// TIA Portal V18 export
// export: Created 2024-02-15T13:16:19.4089202Z, ExportSetting WithDefaults, DisplayName Totally Integrated Automation Portal, DisplayVersion V18 Update 3, DisplayName TIA Portal Openness, DisplayVersion V18 Update 3, DisplayName TIA Portal Version Control Interface, DisplayVersion V18, DisplayName TIA Portal Test Suite Advanced, DisplayVersion V18, DisplayName SINAMICS Startdrive Advanced, DisplayVersion V18, DisplayName SINAMICS Startdrive G130, G150, S120, S150, SINAMICS MV, S210, DisplayVersion V18, DisplayName SINAMICS Startdrive G110M, G120, G120C, G120D, G120P, G115D, DisplayVersion V18, DisplayName STEP 7 Professional, DisplayVersion V18 Update 3, DisplayName STEP 7 CFC, DisplayVersion V18, DisplayName STEP 7 Safety, DisplayVersion V18, DisplayName WinCC Advanced / Unified PC, DisplayVersion V18 Update 3, DisplayName SIMATIC Visualization Architect, DisplayVersion V18 Update 3
FUNCTION "COM_8864079" : Void   // FC36, LAD
{ S7_Optimized_Access := 'TRUE' }
VERSION : 0.1
// stored: AutoNumber true, IsIECCheckEnabled false, SetENOAutomatically false, UDAEnableTagReadback false
   VAR_TEMP   // added for the SCL form of the ladder/FBD networks
      _w1 : Bool;
   END_VAR
BEGIN

REGION Network 1: Echange avec API SDM Demande de Froid
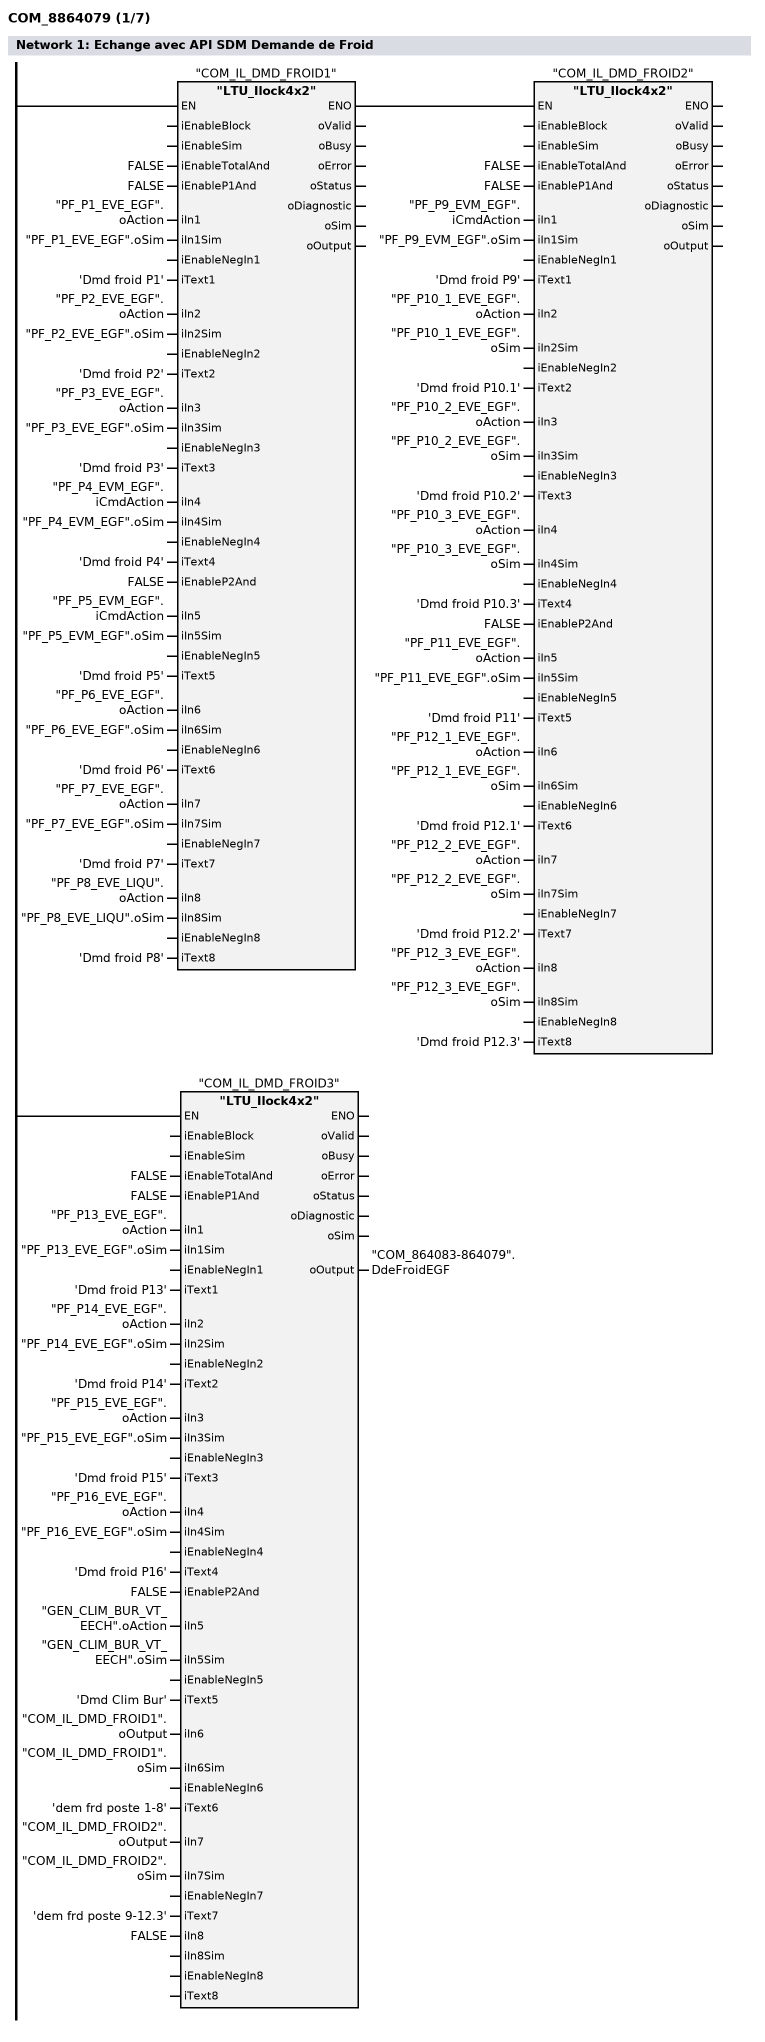
   RUNG wire#powerrail
      "COM_IL_DMD_FROID1"(iEnableBlock :=, iEnableSim :=, iEnableTotalAnd := FALSE, iEnableP1And := FALSE, iIn1 := "PF_P1_EVE_EGF".oAction, iIn1Sim := "PF_P1_EVE_EGF".oSim, iEnableNegIn1 :=, iText1 := 'Dmd froid P1', iIn2 := "PF_P2_EVE_EGF".oAction, iIn2Sim := "PF_P2_EVE_EGF".oSim, iEnableNegIn2 :=, iText2 := 'Dmd froid P2', iIn3 := "PF_P3_EVE_EGF".oAction, iIn3Sim := "PF_P3_EVE_EGF".oSim, iEnableNegIn3 :=, iText3 := 'Dmd froid P3', iIn4 := "PF_P4_EVM_EGF".iCmdAction, iIn4Sim := "PF_P4_EVM_EGF".oSim, iEnableNegIn4 :=, iText4 := 'Dmd froid P4', iEnableP2And := FALSE, iIn5 := "PF_P5_EVM_EGF".iCmdAction, iIn5Sim := "PF_P5_EVM_EGF".oSim, iEnableNegIn5 :=, iText5 := 'Dmd froid P5', iIn6 := "PF_P6_EVE_EGF".oAction, iIn6Sim := "PF_P6_EVE_EGF".oSim, iEnableNegIn6 :=, iText6 := 'Dmd froid P6', iIn7 := "PF_P7_EVE_EGF".oAction, iIn7Sim := "PF_P7_EVE_EGF".oSim, iEnableNegIn7 :=, iText7 := 'Dmd froid P7', iIn8 := "PF_P8_EVE_LIQU".oAction, iIn8Sim := "PF_P8_EVE_LIQU".oSim, iEnableNegIn8 :=, iText8 := 'Dmd froid P8', oValid =>, oBusy =>, oError =>, oStatus =>, oDiagnostic =>, oSim =>, oOutput =>)
      "COM_IL_DMD_FROID2"(iEnableBlock :=, iEnableSim :=, iEnableTotalAnd := FALSE, iEnableP1And := FALSE, iIn1 := "PF_P9_EVM_EGF".iCmdAction, iIn1Sim := "PF_P9_EVM_EGF".oSim, iEnableNegIn1 :=, iText1 := 'Dmd froid P9', iIn2 := "PF_P10_1_EVE_EGF".oAction, iIn2Sim := "PF_P10_1_EVE_EGF".oSim, iEnableNegIn2 :=, iText2 := 'Dmd froid P10.1', iIn3 := "PF_P10_2_EVE_EGF".oAction, iIn3Sim := "PF_P10_2_EVE_EGF".oSim, iEnableNegIn3 :=, iText3 := 'Dmd froid P10.2', iIn4 := "PF_P10_3_EVE_EGF".oAction, iIn4Sim := "PF_P10_3_EVE_EGF".oSim, iEnableNegIn4 :=, iText4 := 'Dmd froid P10.3', iEnableP2And := FALSE, iIn5 := "PF_P11_EVE_EGF".oAction, iIn5Sim := "PF_P11_EVE_EGF".oSim, iEnableNegIn5 :=, iText5 := 'Dmd froid P11', iIn6 := "PF_P12_1_EVE_EGF".oAction, iIn6Sim := "PF_P12_1_EVE_EGF".oSim, iEnableNegIn6 :=, iText6 := 'Dmd froid P12.1', iIn7 := "PF_P12_2_EVE_EGF".oAction, iIn7Sim := "PF_P12_2_EVE_EGF".oSim, iEnableNegIn7 :=, iText7 := 'Dmd froid P12.2', iIn8 := "PF_P12_3_EVE_EGF".oAction, iIn8Sim := "PF_P12_3_EVE_EGF".oSim, iEnableNegIn8 :=, iText8 := 'Dmd froid P12.3', oValid =>, oBusy =>, oError =>, oStatus =>, oDiagnostic =>, oSim =>, oOutput =>)
   END_RUNG
   RUNG wire#powerrail
      "COM_IL_DMD_FROID3"(iEnableBlock :=, iEnableSim :=, iEnableTotalAnd := FALSE, iEnableP1And := FALSE, iIn1 := "PF_P13_EVE_EGF".oAction, iIn1Sim := "PF_P13_EVE_EGF".oSim, iEnableNegIn1 :=, iText1 := 'Dmd froid P13', iIn2 := "PF_P14_EVE_EGF".oAction, iIn2Sim := "PF_P14_EVE_EGF".oSim, iEnableNegIn2 :=, iText2 := 'Dmd froid P14', iIn3 := "PF_P15_EVE_EGF".oAction, iIn3Sim := "PF_P15_EVE_EGF".oSim, iEnableNegIn3 :=, iText3 := 'Dmd froid P15', iIn4 := "PF_P16_EVE_EGF".oAction, iIn4Sim := "PF_P16_EVE_EGF".oSim, iEnableNegIn4 :=, iText4 := 'Dmd froid P16', iEnableP2And := FALSE, iIn5 := "GEN_CLIM_BUR_VT_EECH".oAction, iIn5Sim := "GEN_CLIM_BUR_VT_EECH".oSim, iEnableNegIn5 :=, iText5 := 'Dmd Clim Bur', iIn6 := "COM_IL_DMD_FROID1".oOutput, iIn6Sim := "COM_IL_DMD_FROID1".oSim, iEnableNegIn6 :=, iText6 := 'dem frd poste 1-8', iIn7 := "COM_IL_DMD_FROID2".oOutput, iIn7Sim := "COM_IL_DMD_FROID2".oSim, iEnableNegIn7 :=, iText7 := 'dem frd poste 9-12.3', iIn8 := FALSE, iIn8Sim :=, iEnableNegIn8 :=, iText8 :=, oValid =>, oBusy =>, oError =>, oStatus =>, oDiagnostic =>, oSim =>, oOutput => "COM_864083-864079".DdeFroidEGF)
   END_RUNG
   // the same network as SCL:
   "COM_IL_DMD_FROID1"(iEnableTotalAnd := FALSE,   // "LTU_Ilock4x2"
                       iEnableP1And := FALSE,
                       iIn1 := "PF_P1_EVE_EGF".oAction,
                       iIn1Sim := "PF_P1_EVE_EGF".oSim,
                       iText1 := 'Dmd froid P1',
                       iIn2 := "PF_P2_EVE_EGF".oAction,
                       iIn2Sim := "PF_P2_EVE_EGF".oSim,
                       iText2 := 'Dmd froid P2',
                       iIn3 := "PF_P3_EVE_EGF".oAction,
                       iIn3Sim := "PF_P3_EVE_EGF".oSim,
                       iText3 := 'Dmd froid P3',
                       iIn4 := "PF_P4_EVM_EGF".iCmdAction,
                       iIn4Sim := "PF_P4_EVM_EGF".oSim,
                       iText4 := 'Dmd froid P4',
                       iEnableP2And := FALSE,
                       iIn5 := "PF_P5_EVM_EGF".iCmdAction,
                       iIn5Sim := "PF_P5_EVM_EGF".oSim,
                       iText5 := 'Dmd froid P5',
                       iIn6 := "PF_P6_EVE_EGF".oAction,
                       iIn6Sim := "PF_P6_EVE_EGF".oSim,
                       iText6 := 'Dmd froid P6',
                       iIn7 := "PF_P7_EVE_EGF".oAction,
                       iIn7Sim := "PF_P7_EVE_EGF".oSim,
                       iText7 := 'Dmd froid P7',
                       iIn8 := "PF_P8_EVE_LIQU".oAction,
                       iIn8Sim := "PF_P8_EVE_LIQU".oSim,
                       iText8 := 'Dmd froid P8',
                       ENO => #_w1);
   IF #_w1 THEN
       "COM_IL_DMD_FROID2"(iEnableTotalAnd := FALSE,   // "LTU_Ilock4x2"
                           iEnableP1And := FALSE,
                           iIn1 := "PF_P9_EVM_EGF".iCmdAction,
                           iIn1Sim := "PF_P9_EVM_EGF".oSim,
                           iText1 := 'Dmd froid P9',
                           iIn2 := "PF_P10_1_EVE_EGF".oAction,
                           iIn2Sim := "PF_P10_1_EVE_EGF".oSim,
                           iText2 := 'Dmd froid P10.1',
                           iIn3 := "PF_P10_2_EVE_EGF".oAction,
                           iIn3Sim := "PF_P10_2_EVE_EGF".oSim,
                           iText3 := 'Dmd froid P10.2',
                           iIn4 := "PF_P10_3_EVE_EGF".oAction,
                           iIn4Sim := "PF_P10_3_EVE_EGF".oSim,
                           iText4 := 'Dmd froid P10.3',
                           iEnableP2And := FALSE,
                           iIn5 := "PF_P11_EVE_EGF".oAction,
                           iIn5Sim := "PF_P11_EVE_EGF".oSim,
                           iText5 := 'Dmd froid P11',
                           iIn6 := "PF_P12_1_EVE_EGF".oAction,
                           iIn6Sim := "PF_P12_1_EVE_EGF".oSim,
                           iText6 := 'Dmd froid P12.1',
                           iIn7 := "PF_P12_2_EVE_EGF".oAction,
                           iIn7Sim := "PF_P12_2_EVE_EGF".oSim,
                           iText7 := 'Dmd froid P12.2',
                           iIn8 := "PF_P12_3_EVE_EGF".oAction,
                           iIn8Sim := "PF_P12_3_EVE_EGF".oSim,
                           iText8 := 'Dmd froid P12.3');
   END_IF;
   "COM_IL_DMD_FROID3"(iEnableTotalAnd := FALSE,   // "LTU_Ilock4x2"
                       iEnableP1And := FALSE,
                       iIn1 := "PF_P13_EVE_EGF".oAction,
                       iIn1Sim := "PF_P13_EVE_EGF".oSim,
                       iText1 := 'Dmd froid P13',
                       iIn2 := "PF_P14_EVE_EGF".oAction,
                       iIn2Sim := "PF_P14_EVE_EGF".oSim,
                       iText2 := 'Dmd froid P14',
                       iIn3 := "PF_P15_EVE_EGF".oAction,
                       iIn3Sim := "PF_P15_EVE_EGF".oSim,
                       iText3 := 'Dmd froid P15',
                       iIn4 := "PF_P16_EVE_EGF".oAction,
                       iIn4Sim := "PF_P16_EVE_EGF".oSim,
                       iText4 := 'Dmd froid P16',
                       iEnableP2And := FALSE,
                       iIn5 := "GEN_CLIM_BUR_VT_EECH".oAction,
                       iIn5Sim := "GEN_CLIM_BUR_VT_EECH".oSim,
                       iText5 := 'Dmd Clim Bur',
                       iIn6 := "COM_IL_DMD_FROID1".oOutput,
                       iIn6Sim := "COM_IL_DMD_FROID1".oSim,
                       iText6 := 'dem frd poste 1-8',
                       iIn7 := "COM_IL_DMD_FROID2".oOutput,
                       iIn7Sim := "COM_IL_DMD_FROID2".oSim,
                       iText7 := 'dem frd poste 9-12.3',
                       iIn8 := FALSE,
                       oOutput => "COM_864083-864079".DdeFroidEGF);
END_REGION

REGION Network 2: Echange avec API SDM Demande de Dégivrage
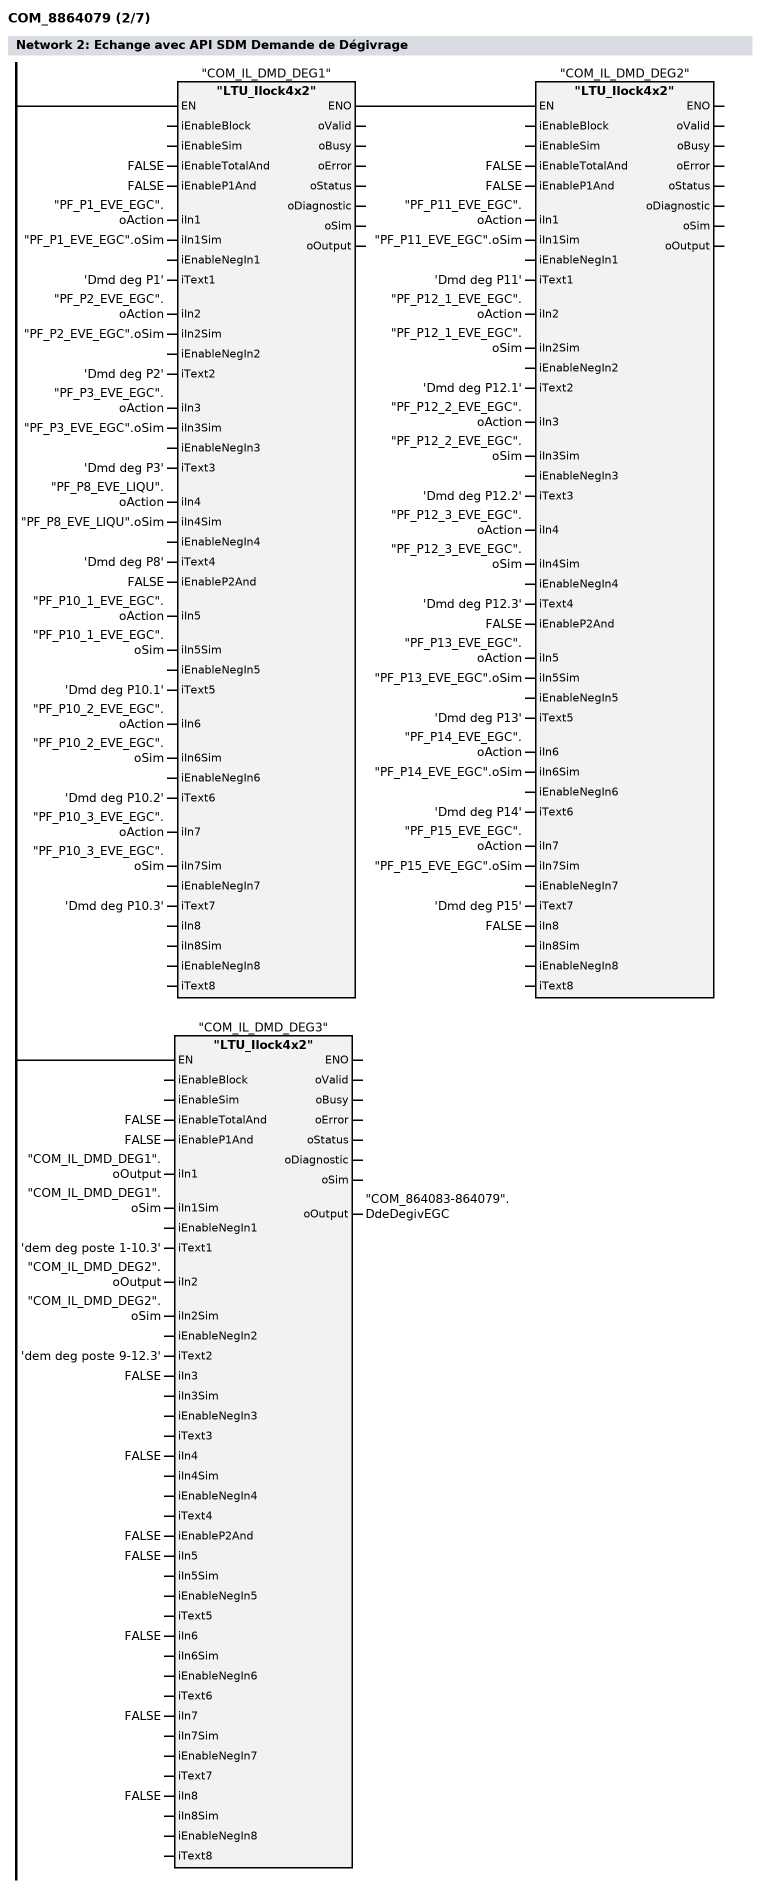
   RUNG wire#powerrail
      "COM_IL_DMD_DEG1"(iEnableBlock :=, iEnableSim :=, iEnableTotalAnd := FALSE, iEnableP1And := FALSE, iIn1 := "PF_P1_EVE_EGC".oAction, iIn1Sim := "PF_P1_EVE_EGC".oSim, iEnableNegIn1 :=, iText1 := 'Dmd deg P1', iIn2 := "PF_P2_EVE_EGC".oAction, iIn2Sim := "PF_P2_EVE_EGC".oSim, iEnableNegIn2 :=, iText2 := 'Dmd deg P2', iIn3 := "PF_P3_EVE_EGC".oAction, iIn3Sim := "PF_P3_EVE_EGC".oSim, iEnableNegIn3 :=, iText3 := 'Dmd deg P3', iIn4 := "PF_P8_EVE_LIQU".oAction, iIn4Sim := "PF_P8_EVE_LIQU".oSim, iEnableNegIn4 :=, iText4 := 'Dmd deg P8', iEnableP2And := FALSE, iIn5 := "PF_P10_1_EVE_EGC".oAction, iIn5Sim := "PF_P10_1_EVE_EGC".oSim, iEnableNegIn5 :=, iText5 := 'Dmd deg P10.1', iIn6 := "PF_P10_2_EVE_EGC".oAction, iIn6Sim := "PF_P10_2_EVE_EGC".oSim, iEnableNegIn6 :=, iText6 := 'Dmd deg P10.2', iIn7 := "PF_P10_3_EVE_EGC".oAction, iIn7Sim := "PF_P10_3_EVE_EGC".oSim, iEnableNegIn7 :=, iText7 := 'Dmd deg P10.3', iIn8 :=, iIn8Sim :=, iEnableNegIn8 :=, iText8 :=, oValid =>, oBusy =>, oError =>, oStatus =>, oDiagnostic =>, oSim =>, oOutput =>)
      "COM_IL_DMD_DEG2"(iEnableBlock :=, iEnableSim :=, iEnableTotalAnd := FALSE, iEnableP1And := FALSE, iIn1 := "PF_P11_EVE_EGC".oAction, iIn1Sim := "PF_P11_EVE_EGC".oSim, iEnableNegIn1 :=, iText1 := 'Dmd deg P11', iIn2 := "PF_P12_1_EVE_EGC".oAction, iIn2Sim := "PF_P12_1_EVE_EGC".oSim, iEnableNegIn2 :=, iText2 := 'Dmd deg P12.1', iIn3 := "PF_P12_2_EVE_EGC".oAction, iIn3Sim := "PF_P12_2_EVE_EGC".oSim, iEnableNegIn3 :=, iText3 := 'Dmd deg P12.2', iIn4 := "PF_P12_3_EVE_EGC".oAction, iIn4Sim := "PF_P12_3_EVE_EGC".oSim, iEnableNegIn4 :=, iText4 := 'Dmd deg P12.3', iEnableP2And := FALSE, iIn5 := "PF_P13_EVE_EGC".oAction, iIn5Sim := "PF_P13_EVE_EGC".oSim, iEnableNegIn5 :=, iText5 := 'Dmd deg P13', iIn6 := "PF_P14_EVE_EGC".oAction, iIn6Sim := "PF_P14_EVE_EGC".oSim, iEnableNegIn6 :=, iText6 := 'Dmd deg P14', iIn7 := "PF_P15_EVE_EGC".oAction, iIn7Sim := "PF_P15_EVE_EGC".oSim, iEnableNegIn7 :=, iText7 := 'Dmd deg P15', iIn8 := FALSE, iIn8Sim :=, iEnableNegIn8 :=, iText8 :=, oValid =>, oBusy =>, oError =>, oStatus =>, oDiagnostic =>, oSim =>, oOutput =>)
   END_RUNG
   RUNG wire#powerrail
      "COM_IL_DMD_DEG3"(iEnableBlock :=, iEnableSim :=, iEnableTotalAnd := FALSE, iEnableP1And := FALSE, iIn1 := "COM_IL_DMD_DEG1".oOutput, iIn1Sim := "COM_IL_DMD_DEG1".oSim, iEnableNegIn1 :=, iText1 := 'dem deg poste 1-10.3', iIn2 := "COM_IL_DMD_DEG2".oOutput, iIn2Sim := "COM_IL_DMD_DEG2".oSim, iEnableNegIn2 :=, iText2 := 'dem deg poste 9-12.3', iIn3 := FALSE, iIn3Sim :=, iEnableNegIn3 :=, iText3 :=, iIn4 := FALSE, iIn4Sim :=, iEnableNegIn4 :=, iText4 :=, iEnableP2And := FALSE, iIn5 := FALSE, iIn5Sim :=, iEnableNegIn5 :=, iText5 :=, iIn6 := FALSE, iIn6Sim :=, iEnableNegIn6 :=, iText6 :=, iIn7 := FALSE, iIn7Sim :=, iEnableNegIn7 :=, iText7 :=, iIn8 := FALSE, iIn8Sim :=, iEnableNegIn8 :=, iText8 :=, oValid =>, oBusy =>, oError =>, oStatus =>, oDiagnostic =>, oSim =>, oOutput => "COM_864083-864079".DdeDegivEGC)
   END_RUNG
   // the same network as SCL:
   "COM_IL_DMD_DEG1"(iEnableTotalAnd := FALSE,   // "LTU_Ilock4x2"
                     iEnableP1And := FALSE,
                     iIn1 := "PF_P1_EVE_EGC".oAction,
                     iIn1Sim := "PF_P1_EVE_EGC".oSim,
                     iText1 := 'Dmd deg P1',
                     iIn2 := "PF_P2_EVE_EGC".oAction,
                     iIn2Sim := "PF_P2_EVE_EGC".oSim,
                     iText2 := 'Dmd deg P2',
                     iIn3 := "PF_P3_EVE_EGC".oAction,
                     iIn3Sim := "PF_P3_EVE_EGC".oSim,
                     iText3 := 'Dmd deg P3',
                     iIn4 := "PF_P8_EVE_LIQU".oAction,
                     iIn4Sim := "PF_P8_EVE_LIQU".oSim,
                     iText4 := 'Dmd deg P8',
                     iEnableP2And := FALSE,
                     iIn5 := "PF_P10_1_EVE_EGC".oAction,
                     iIn5Sim := "PF_P10_1_EVE_EGC".oSim,
                     iText5 := 'Dmd deg P10.1',
                     iIn6 := "PF_P10_2_EVE_EGC".oAction,
                     iIn6Sim := "PF_P10_2_EVE_EGC".oSim,
                     iText6 := 'Dmd deg P10.2',
                     iIn7 := "PF_P10_3_EVE_EGC".oAction,
                     iIn7Sim := "PF_P10_3_EVE_EGC".oSim,
                     iText7 := 'Dmd deg P10.3',
                     ENO => #_w1);
   IF #_w1 THEN
       "COM_IL_DMD_DEG2"(iEnableTotalAnd := FALSE,   // "LTU_Ilock4x2"
                         iEnableP1And := FALSE,
                         iIn1 := "PF_P11_EVE_EGC".oAction,
                         iIn1Sim := "PF_P11_EVE_EGC".oSim,
                         iText1 := 'Dmd deg P11',
                         iIn2 := "PF_P12_1_EVE_EGC".oAction,
                         iIn2Sim := "PF_P12_1_EVE_EGC".oSim,
                         iText2 := 'Dmd deg P12.1',
                         iIn3 := "PF_P12_2_EVE_EGC".oAction,
                         iIn3Sim := "PF_P12_2_EVE_EGC".oSim,
                         iText3 := 'Dmd deg P12.2',
                         iIn4 := "PF_P12_3_EVE_EGC".oAction,
                         iIn4Sim := "PF_P12_3_EVE_EGC".oSim,
                         iText4 := 'Dmd deg P12.3',
                         iEnableP2And := FALSE,
                         iIn5 := "PF_P13_EVE_EGC".oAction,
                         iIn5Sim := "PF_P13_EVE_EGC".oSim,
                         iText5 := 'Dmd deg P13',
                         iIn6 := "PF_P14_EVE_EGC".oAction,
                         iIn6Sim := "PF_P14_EVE_EGC".oSim,
                         iText6 := 'Dmd deg P14',
                         iIn7 := "PF_P15_EVE_EGC".oAction,
                         iIn7Sim := "PF_P15_EVE_EGC".oSim,
                         iText7 := 'Dmd deg P15',
                         iIn8 := FALSE);
   END_IF;
   "COM_IL_DMD_DEG3"(iEnableTotalAnd := FALSE,   // "LTU_Ilock4x2"
                     iEnableP1And := FALSE,
                     iIn1 := "COM_IL_DMD_DEG1".oOutput,
                     iIn1Sim := "COM_IL_DMD_DEG1".oSim,
                     iText1 := 'dem deg poste 1-10.3',
                     iIn2 := "COM_IL_DMD_DEG2".oOutput,
                     iIn2Sim := "COM_IL_DMD_DEG2".oSim,
                     iText2 := 'dem deg poste 9-12.3',
                     iIn3 := FALSE,
                     iIn4 := FALSE,
                     iEnableP2And := FALSE,
                     iIn5 := FALSE,
                     iIn6 := FALSE,
                     iIn7 := FALSE,
                     iIn8 := FALSE,
                     oOutput => "COM_864083-864079".DdeDegivEGC);
END_REGION

REGION Network 3: Echange avec API SDM Défaut prioritaire AGBT1
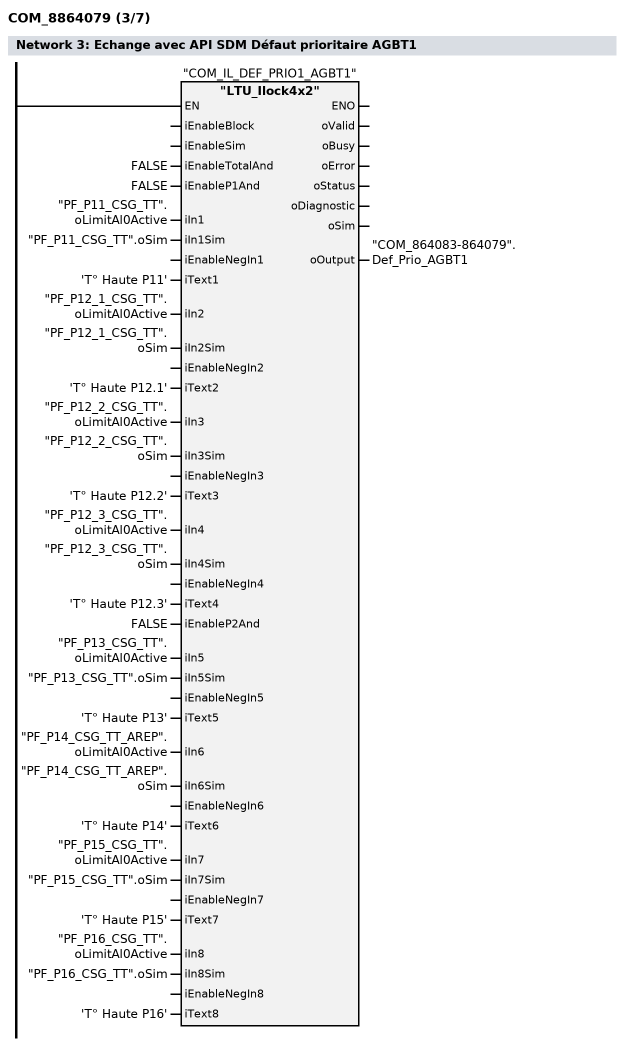
   RUNG wire#powerrail
      "COM_IL_DEF_PRIO1_AGBT1"(iEnableBlock :=, iEnableSim :=, iEnableTotalAnd := FALSE, iEnableP1And := FALSE, iIn1 := "PF_P11_CSG_TT".oLimitAl0Active, iIn1Sim := "PF_P11_CSG_TT".oSim, iEnableNegIn1 :=, iText1 := 'T° Haute P11', iIn2 := "PF_P12_1_CSG_TT".oLimitAl0Active, iIn2Sim := "PF_P12_1_CSG_TT".oSim, iEnableNegIn2 :=, iText2 := 'T° Haute P12.1', iIn3 := "PF_P12_2_CSG_TT".oLimitAl0Active, iIn3Sim := "PF_P12_2_CSG_TT".oSim, iEnableNegIn3 :=, iText3 := 'T° Haute P12.2', iIn4 := "PF_P12_3_CSG_TT".oLimitAl0Active, iIn4Sim := "PF_P12_3_CSG_TT".oSim, iEnableNegIn4 :=, iText4 := 'T° Haute P12.3', iEnableP2And := FALSE, iIn5 := "PF_P13_CSG_TT".oLimitAl0Active, iIn5Sim := "PF_P13_CSG_TT".oSim, iEnableNegIn5 :=, iText5 := 'T° Haute P13', iIn6 := "PF_P14_CSG_TT_AREP".oLimitAl0Active, iIn6Sim := "PF_P14_CSG_TT_AREP".oSim, iEnableNegIn6 :=, iText6 := 'T° Haute P14', iIn7 := "PF_P15_CSG_TT".oLimitAl0Active, iIn7Sim := "PF_P15_CSG_TT".oSim, iEnableNegIn7 :=, iText7 := 'T° Haute P15', iIn8 := "PF_P16_CSG_TT".oLimitAl0Active, iIn8Sim := "PF_P16_CSG_TT".oSim, iEnableNegIn8 :=, iText8 := 'T° Haute P16', oValid =>, oBusy =>, oError =>, oStatus =>, oDiagnostic =>, oSim =>, oOutput => "COM_864083-864079".Def_Prio_AGBT1)
   END_RUNG
   // the same network as SCL:
   "COM_IL_DEF_PRIO1_AGBT1"(iEnableTotalAnd := FALSE,   // "LTU_Ilock4x2"
                           iEnableP1And := FALSE,
                           iIn1 := "PF_P11_CSG_TT".oLimitAl0Active,
                           iIn1Sim := "PF_P11_CSG_TT".oSim,
                           iText1 := 'T° Haute P11',
                           iIn2 := "PF_P12_1_CSG_TT".oLimitAl0Active,
                           iIn2Sim := "PF_P12_1_CSG_TT".oSim,
                           iText2 := 'T° Haute P12.1',
                           iIn3 := "PF_P12_2_CSG_TT".oLimitAl0Active,
                           iIn3Sim := "PF_P12_2_CSG_TT".oSim,
                           iText3 := 'T° Haute P12.2',
                           iIn4 := "PF_P12_3_CSG_TT".oLimitAl0Active,
                           iIn4Sim := "PF_P12_3_CSG_TT".oSim,
                           iText4 := 'T° Haute P12.3',
                           iEnableP2And := FALSE,
                           iIn5 := "PF_P13_CSG_TT".oLimitAl0Active,
                           iIn5Sim := "PF_P13_CSG_TT".oSim,
                           iText5 := 'T° Haute P13',
                           iIn6 := "PF_P14_CSG_TT_AREP".oLimitAl0Active,
                           iIn6Sim := "PF_P14_CSG_TT_AREP".oSim,
                           iText6 := 'T° Haute P14',
                           iIn7 := "PF_P15_CSG_TT".oLimitAl0Active,
                           iIn7Sim := "PF_P15_CSG_TT".oSim,
                           iText7 := 'T° Haute P15',
                           iIn8 := "PF_P16_CSG_TT".oLimitAl0Active,
                           iIn8Sim := "PF_P16_CSG_TT".oSim,
                           iText8 := 'T° Haute P16',
                           oOutput => "COM_864083-864079".Def_Prio_AGBT1);
END_REGION

REGION Network 4: Echange avec API SDM Défaut NON prioritaire AGBT1
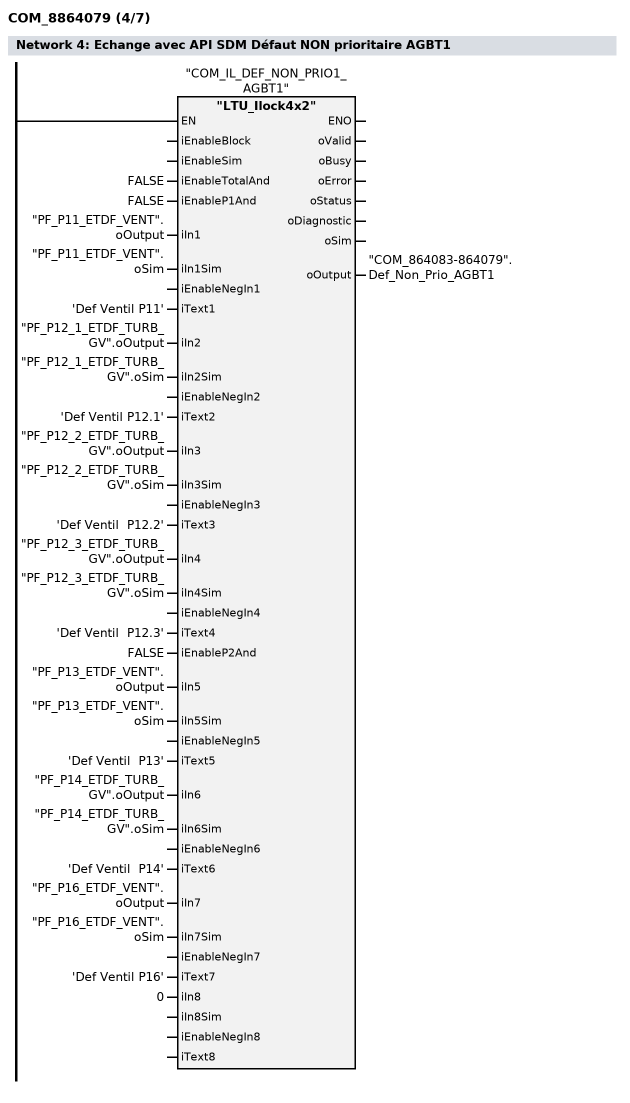
   RUNG wire#powerrail
      "COM_IL_DEF_NON_PRIO1_AGBT1"(iEnableBlock :=, iEnableSim :=, iEnableTotalAnd := FALSE, iEnableP1And := FALSE, iIn1 := "PF_P11_ETDF_VENT".oOutput, iIn1Sim := "PF_P11_ETDF_VENT".oSim, iEnableNegIn1 :=, iText1 := 'Def Ventil P11', iIn2 := "PF_P12_1_ETDF_TURB_GV".oOutput, iIn2Sim := "PF_P12_1_ETDF_TURB_GV".oSim, iEnableNegIn2 :=, iText2 := 'Def Ventil P12.1', iIn3 := "PF_P12_2_ETDF_TURB_GV".oOutput, iIn3Sim := "PF_P12_2_ETDF_TURB_GV".oSim, iEnableNegIn3 :=, iText3 := 'Def Ventil  P12.2', iIn4 := "PF_P12_3_ETDF_TURB_GV".oOutput, iIn4Sim := "PF_P12_3_ETDF_TURB_GV".oSim, iEnableNegIn4 :=, iText4 := 'Def Ventil  P12.3', iEnableP2And := FALSE, iIn5 := "PF_P13_ETDF_VENT".oOutput, iIn5Sim := "PF_P13_ETDF_VENT".oSim, iEnableNegIn5 :=, iText5 := 'Def Ventil  P13', iIn6 := "PF_P14_ETDF_TURB_GV".oOutput, iIn6Sim := "PF_P14_ETDF_TURB_GV".oSim, iEnableNegIn6 :=, iText6 := 'Def Ventil  P14', iIn7 := "PF_P16_ETDF_VENT".oOutput, iIn7Sim := "PF_P16_ETDF_VENT".oSim, iEnableNegIn7 :=, iText7 := 'Def Ventil P16', iIn8 := 0, iIn8Sim :=, iEnableNegIn8 :=, iText8 :=, oValid =>, oBusy =>, oError =>, oStatus =>, oDiagnostic =>, oSim =>, oOutput => "COM_864083-864079".Def_Non_Prio_AGBT1)
   END_RUNG
   // the same network as SCL:
   "COM_IL_DEF_NON_PRIO1_AGBT1"(iEnableTotalAnd := FALSE,   // "LTU_Ilock4x2"
                           iEnableP1And := FALSE,
                           iIn1 := "PF_P11_ETDF_VENT".oOutput,
                           iIn1Sim := "PF_P11_ETDF_VENT".oSim,
                           iText1 := 'Def Ventil P11',
                           iIn2 := "PF_P12_1_ETDF_TURB_GV".oOutput,
                           iIn2Sim := "PF_P12_1_ETDF_TURB_GV".oSim,
                           iText2 := 'Def Ventil P12.1',
                           iIn3 := "PF_P12_2_ETDF_TURB_GV".oOutput,
                           iIn3Sim := "PF_P12_2_ETDF_TURB_GV".oSim,
                           iText3 := 'Def Ventil  P12.2',
                           iIn4 := "PF_P12_3_ETDF_TURB_GV".oOutput,
                           iIn4Sim := "PF_P12_3_ETDF_TURB_GV".oSim,
                           iText4 := 'Def Ventil  P12.3',
                           iEnableP2And := FALSE,
                           iIn5 := "PF_P13_ETDF_VENT".oOutput,
                           iIn5Sim := "PF_P13_ETDF_VENT".oSim,
                           iText5 := 'Def Ventil  P13',
                           iIn6 := "PF_P14_ETDF_TURB_GV".oOutput,
                           iIn6Sim := "PF_P14_ETDF_TURB_GV".oSim,
                           iText6 := 'Def Ventil  P14',
                           iIn7 := "PF_P16_ETDF_VENT".oOutput,
                           iIn7Sim := "PF_P16_ETDF_VENT".oSim,
                           iText7 := 'Def Ventil P16',
                           iIn8 := 0,
                           oOutput => "COM_864083-864079".Def_Non_Prio_AGBT1);
END_REGION

REGION Network 5: Echange avec API SDM Défaut prioritaire AGBT2
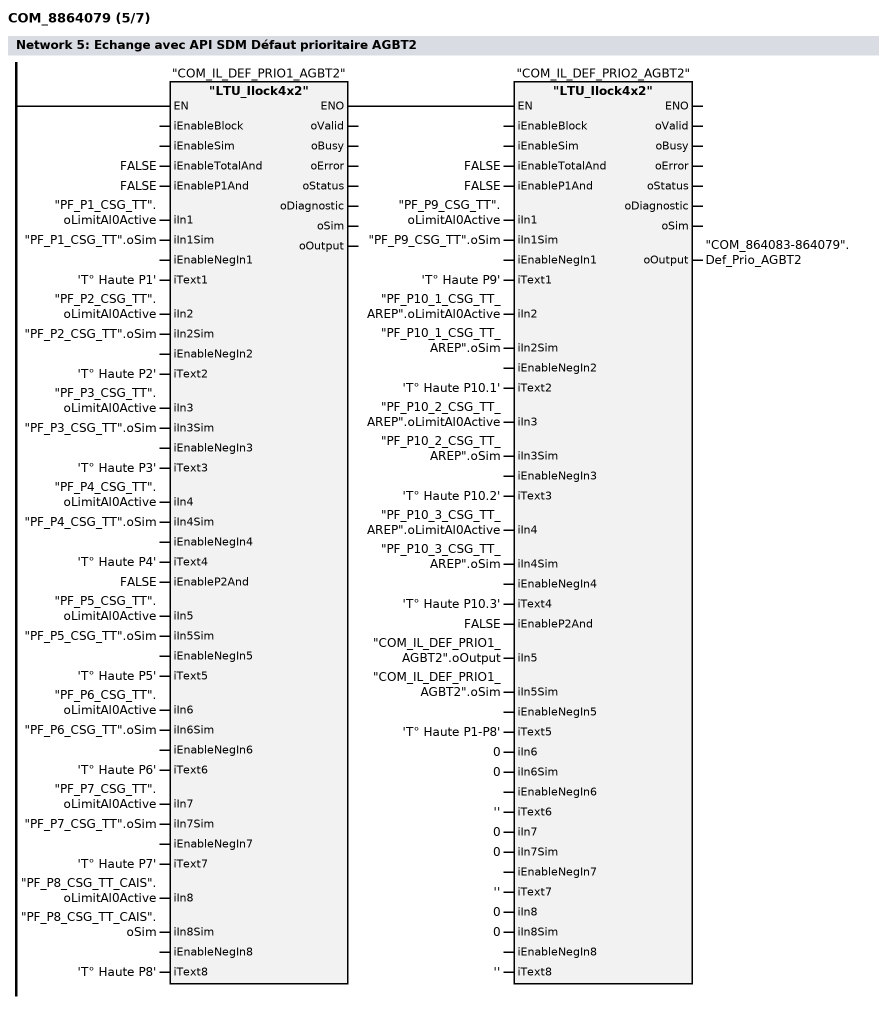
   RUNG wire#powerrail
      "COM_IL_DEF_PRIO1_AGBT2"(iEnableBlock :=, iEnableSim :=, iEnableTotalAnd := FALSE, iEnableP1And := FALSE, iIn1 := "PF_P1_CSG_TT".oLimitAl0Active, iIn1Sim := "PF_P1_CSG_TT".oSim, iEnableNegIn1 :=, iText1 := 'T° Haute P1', iIn2 := "PF_P2_CSG_TT".oLimitAl0Active, iIn2Sim := "PF_P2_CSG_TT".oSim, iEnableNegIn2 :=, iText2 := 'T° Haute P2', iIn3 := "PF_P3_CSG_TT".oLimitAl0Active, iIn3Sim := "PF_P3_CSG_TT".oSim, iEnableNegIn3 :=, iText3 := 'T° Haute P3', iIn4 := "PF_P4_CSG_TT".oLimitAl0Active, iIn4Sim := "PF_P4_CSG_TT".oSim, iEnableNegIn4 :=, iText4 := 'T° Haute P4', iEnableP2And := FALSE, iIn5 := "PF_P5_CSG_TT".oLimitAl0Active, iIn5Sim := "PF_P5_CSG_TT".oSim, iEnableNegIn5 :=, iText5 := 'T° Haute P5', iIn6 := "PF_P6_CSG_TT".oLimitAl0Active, iIn6Sim := "PF_P6_CSG_TT".oSim, iEnableNegIn6 :=, iText6 := 'T° Haute P6', iIn7 := "PF_P7_CSG_TT".oLimitAl0Active, iIn7Sim := "PF_P7_CSG_TT".oSim, iEnableNegIn7 :=, iText7 := 'T° Haute P7', iIn8 := "PF_P8_CSG_TT_CAIS".oLimitAl0Active, iIn8Sim := "PF_P8_CSG_TT_CAIS".oSim, iEnableNegIn8 :=, iText8 := 'T° Haute P8', oValid =>, oBusy =>, oError =>, oStatus =>, oDiagnostic =>, oSim =>, oOutput =>)
      "COM_IL_DEF_PRIO2_AGBT2"(iEnableBlock :=, iEnableSim :=, iEnableTotalAnd := FALSE, iEnableP1And := FALSE, iIn1 := "PF_P9_CSG_TT".oLimitAl0Active, iIn1Sim := "PF_P9_CSG_TT".oSim, iEnableNegIn1 :=, iText1 := 'T° Haute P9', iIn2 := "PF_P10_1_CSG_TT_AREP".oLimitAl0Active, iIn2Sim := "PF_P10_1_CSG_TT_AREP".oSim, iEnableNegIn2 :=, iText2 := 'T° Haute P10.1', iIn3 := "PF_P10_2_CSG_TT_AREP".oLimitAl0Active, iIn3Sim := "PF_P10_2_CSG_TT_AREP".oSim, iEnableNegIn3 :=, iText3 := 'T° Haute P10.2', iIn4 := "PF_P10_3_CSG_TT_AREP".oLimitAl0Active, iIn4Sim := "PF_P10_3_CSG_TT_AREP".oSim, iEnableNegIn4 :=, iText4 := 'T° Haute P10.3', iEnableP2And := FALSE, iIn5 := "COM_IL_DEF_PRIO1_AGBT2".oOutput, iIn5Sim := "COM_IL_DEF_PRIO1_AGBT2".oSim, iEnableNegIn5 :=, iText5 := 'T° Haute P1-P8', iIn6 := 0, iIn6Sim := 0, iEnableNegIn6 :=, iText6 := '', iIn7 := 0, iIn7Sim := 0, iEnableNegIn7 :=, iText7 := '', iIn8 := 0, iIn8Sim := 0, iEnableNegIn8 :=, iText8 := '', oValid =>, oBusy =>, oError =>, oStatus =>, oDiagnostic =>, oSim =>, oOutput => "COM_864083-864079".Def_Prio_AGBT2)
   END_RUNG
   // the same network as SCL:
   "COM_IL_DEF_PRIO1_AGBT2"(iEnableTotalAnd := FALSE,   // "LTU_Ilock4x2"
                           iEnableP1And := FALSE,
                           iIn1 := "PF_P1_CSG_TT".oLimitAl0Active,
                           iIn1Sim := "PF_P1_CSG_TT".oSim,
                           iText1 := 'T° Haute P1',
                           iIn2 := "PF_P2_CSG_TT".oLimitAl0Active,
                           iIn2Sim := "PF_P2_CSG_TT".oSim,
                           iText2 := 'T° Haute P2',
                           iIn3 := "PF_P3_CSG_TT".oLimitAl0Active,
                           iIn3Sim := "PF_P3_CSG_TT".oSim,
                           iText3 := 'T° Haute P3',
                           iIn4 := "PF_P4_CSG_TT".oLimitAl0Active,
                           iIn4Sim := "PF_P4_CSG_TT".oSim,
                           iText4 := 'T° Haute P4',
                           iEnableP2And := FALSE,
                           iIn5 := "PF_P5_CSG_TT".oLimitAl0Active,
                           iIn5Sim := "PF_P5_CSG_TT".oSim,
                           iText5 := 'T° Haute P5',
                           iIn6 := "PF_P6_CSG_TT".oLimitAl0Active,
                           iIn6Sim := "PF_P6_CSG_TT".oSim,
                           iText6 := 'T° Haute P6',
                           iIn7 := "PF_P7_CSG_TT".oLimitAl0Active,
                           iIn7Sim := "PF_P7_CSG_TT".oSim,
                           iText7 := 'T° Haute P7',
                           iIn8 := "PF_P8_CSG_TT_CAIS".oLimitAl0Active,
                           iIn8Sim := "PF_P8_CSG_TT_CAIS".oSim,
                           iText8 := 'T° Haute P8',
                           ENO => #_w1);
   IF #_w1 THEN
       "COM_IL_DEF_PRIO2_AGBT2"(iEnableTotalAnd := FALSE,   // "LTU_Ilock4x2"
                               iEnableP1And := FALSE,
                               iIn1 := "PF_P9_CSG_TT".oLimitAl0Active,
                               iIn1Sim := "PF_P9_CSG_TT".oSim,
                               iText1 := 'T° Haute P9',
                               iIn2 := "PF_P10_1_CSG_TT_AREP".oLimitAl0Active,
                               iIn2Sim := "PF_P10_1_CSG_TT_AREP".oSim,
                               iText2 := 'T° Haute P10.1',
                               iIn3 := "PF_P10_2_CSG_TT_AREP".oLimitAl0Active,
                               iIn3Sim := "PF_P10_2_CSG_TT_AREP".oSim,
                               iText3 := 'T° Haute P10.2',
                               iIn4 := "PF_P10_3_CSG_TT_AREP".oLimitAl0Active,
                               iIn4Sim := "PF_P10_3_CSG_TT_AREP".oSim,
                               iText4 := 'T° Haute P10.3',
                               iEnableP2And := FALSE,
                               iIn5 := "COM_IL_DEF_PRIO1_AGBT2".oOutput,
                               iIn5Sim := "COM_IL_DEF_PRIO1_AGBT2".oSim,
                               iText5 := 'T° Haute P1-P8',
                               iIn6 := 0,
                               iIn6Sim := 0,
                               iText6 := '',
                               iIn7 := 0,
                               iIn7Sim := 0,
                               iText7 := '',
                               iIn8 := 0,
                               iIn8Sim := 0,
                               iText8 := '',
                               oOutput => "COM_864083-864079".Def_Prio_AGBT2);
   END_IF;
END_REGION

REGION Network 6: Echange avec API SDM Défaut NON prioritaire AGBT2
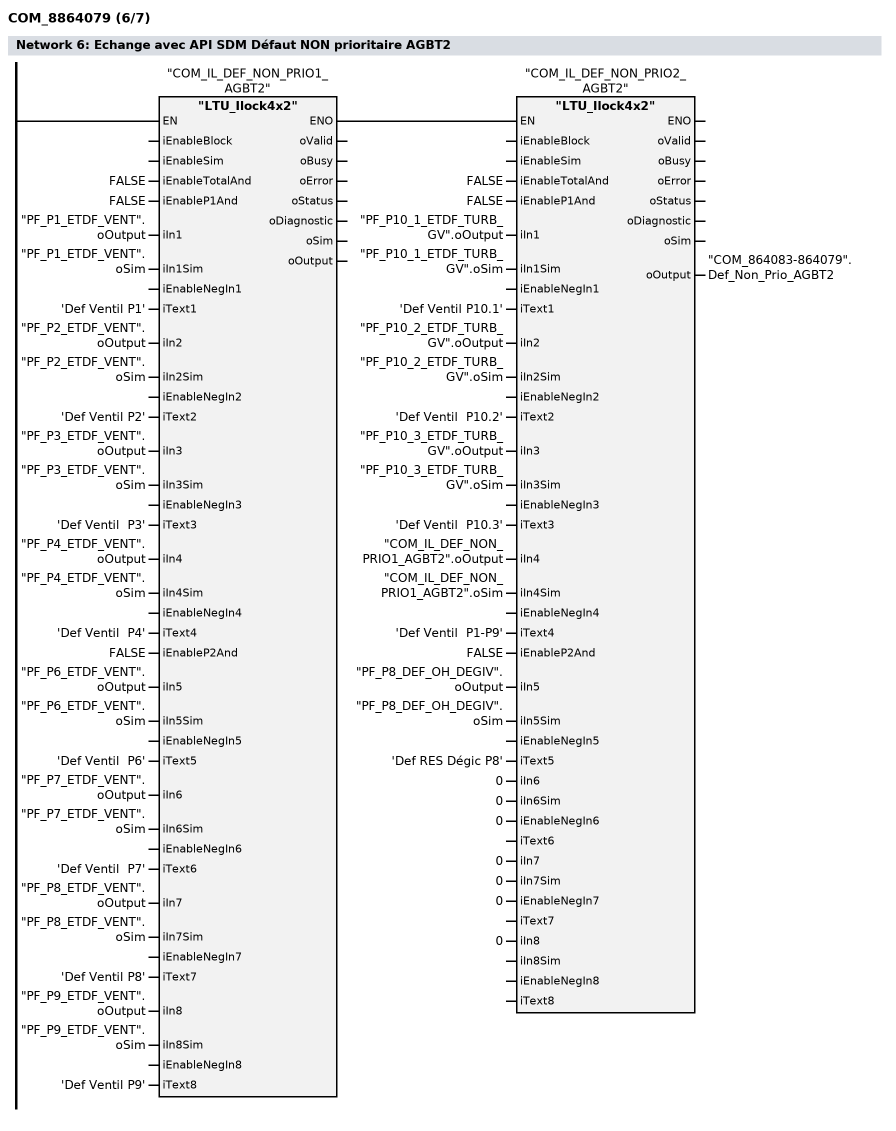
   RUNG wire#powerrail
      "COM_IL_DEF_NON_PRIO1_AGBT2"(iEnableBlock :=, iEnableSim :=, iEnableTotalAnd := FALSE, iEnableP1And := FALSE, iIn1 := "PF_P1_ETDF_VENT".oOutput, iIn1Sim := "PF_P1_ETDF_VENT".oSim, iEnableNegIn1 :=, iText1 := 'Def Ventil P1', iIn2 := "PF_P2_ETDF_VENT".oOutput, iIn2Sim := "PF_P2_ETDF_VENT".oSim, iEnableNegIn2 :=, iText2 := 'Def Ventil P2', iIn3 := "PF_P3_ETDF_VENT".oOutput, iIn3Sim := "PF_P3_ETDF_VENT".oSim, iEnableNegIn3 :=, iText3 := 'Def Ventil  P3', iIn4 := "PF_P4_ETDF_VENT".oOutput, iIn4Sim := "PF_P4_ETDF_VENT".oSim, iEnableNegIn4 :=, iText4 := 'Def Ventil  P4', iEnableP2And := FALSE, iIn5 := "PF_P6_ETDF_VENT".oOutput, iIn5Sim := "PF_P6_ETDF_VENT".oSim, iEnableNegIn5 :=, iText5 := 'Def Ventil  P6', iIn6 := "PF_P7_ETDF_VENT".oOutput, iIn6Sim := "PF_P7_ETDF_VENT".oSim, iEnableNegIn6 :=, iText6 := 'Def Ventil  P7', iIn7 := "PF_P8_ETDF_VENT".oOutput, iIn7Sim := "PF_P8_ETDF_VENT".oSim, iEnableNegIn7 :=, iText7 := 'Def Ventil P8', iIn8 := "PF_P9_ETDF_VENT".oOutput, iIn8Sim := "PF_P9_ETDF_VENT".oSim, iEnableNegIn8 :=, iText8 := 'Def Ventil P9', oValid =>, oBusy =>, oError =>, oStatus =>, oDiagnostic =>, oSim =>, oOutput =>)
      "COM_IL_DEF_NON_PRIO2_AGBT2"(iEnableBlock :=, iEnableSim :=, iEnableTotalAnd := FALSE, iEnableP1And := FALSE, iIn1 := "PF_P10_1_ETDF_TURB_GV".oOutput, iIn1Sim := "PF_P10_1_ETDF_TURB_GV".oSim, iEnableNegIn1 :=, iText1 := 'Def Ventil P10.1', iIn2 := "PF_P10_2_ETDF_TURB_GV".oOutput, iIn2Sim := "PF_P10_2_ETDF_TURB_GV".oSim, iEnableNegIn2 :=, iText2 := 'Def Ventil  P10.2', iIn3 := "PF_P10_3_ETDF_TURB_GV".oOutput, iIn3Sim := "PF_P10_3_ETDF_TURB_GV".oSim, iEnableNegIn3 :=, iText3 := 'Def Ventil  P10.3', iIn4 := "COM_IL_DEF_NON_PRIO1_AGBT2".oOutput, iIn4Sim := "COM_IL_DEF_NON_PRIO1_AGBT2".oSim, iEnableNegIn4 :=, iText4 := 'Def Ventil  P1-P9', iEnableP2And := FALSE, iIn5 := "PF_P8_DEF_OH_DEGIV".oOutput, iIn5Sim := "PF_P8_DEF_OH_DEGIV".oSim, iEnableNegIn5 :=, iText5 := 'Def RES Dégic P8', iIn6 := 0, iIn6Sim := 0, iEnableNegIn6 := 0, iText6 :=, iIn7 := 0, iIn7Sim := 0, iEnableNegIn7 := 0, iText7 :=, iIn8 := 0, iIn8Sim :=, iEnableNegIn8 :=, iText8 :=, oValid =>, oBusy =>, oError =>, oStatus =>, oDiagnostic =>, oSim =>, oOutput => "COM_864083-864079".Def_Non_Prio_AGBT2)
   END_RUNG
   // the same network as SCL:
   "COM_IL_DEF_NON_PRIO1_AGBT2"(iEnableTotalAnd := FALSE,   // "LTU_Ilock4x2"
                           iEnableP1And := FALSE,
                           iIn1 := "PF_P1_ETDF_VENT".oOutput,
                           iIn1Sim := "PF_P1_ETDF_VENT".oSim,
                           iText1 := 'Def Ventil P1',
                           iIn2 := "PF_P2_ETDF_VENT".oOutput,
                           iIn2Sim := "PF_P2_ETDF_VENT".oSim,
                           iText2 := 'Def Ventil P2',
                           iIn3 := "PF_P3_ETDF_VENT".oOutput,
                           iIn3Sim := "PF_P3_ETDF_VENT".oSim,
                           iText3 := 'Def Ventil  P3',
                           iIn4 := "PF_P4_ETDF_VENT".oOutput,
                           iIn4Sim := "PF_P4_ETDF_VENT".oSim,
                           iText4 := 'Def Ventil  P4',
                           iEnableP2And := FALSE,
                           iIn5 := "PF_P6_ETDF_VENT".oOutput,
                           iIn5Sim := "PF_P6_ETDF_VENT".oSim,
                           iText5 := 'Def Ventil  P6',
                           iIn6 := "PF_P7_ETDF_VENT".oOutput,
                           iIn6Sim := "PF_P7_ETDF_VENT".oSim,
                           iText6 := 'Def Ventil  P7',
                           iIn7 := "PF_P8_ETDF_VENT".oOutput,
                           iIn7Sim := "PF_P8_ETDF_VENT".oSim,
                           iText7 := 'Def Ventil P8',
                           iIn8 := "PF_P9_ETDF_VENT".oOutput,
                           iIn8Sim := "PF_P9_ETDF_VENT".oSim,
                           iText8 := 'Def Ventil P9',
                           ENO => #_w1);
   IF #_w1 THEN
       "COM_IL_DEF_NON_PRIO2_AGBT2"(iEnableTotalAnd := FALSE,   // "LTU_Ilock4x2"
                               iEnableP1And := FALSE,
                               iIn1 := "PF_P10_1_ETDF_TURB_GV".oOutput,
                               iIn1Sim := "PF_P10_1_ETDF_TURB_GV".oSim,
                               iText1 := 'Def Ventil P10.1',
                               iIn2 := "PF_P10_2_ETDF_TURB_GV".oOutput,
                               iIn2Sim := "PF_P10_2_ETDF_TURB_GV".oSim,
                               iText2 := 'Def Ventil  P10.2',
                               iIn3 := "PF_P10_3_ETDF_TURB_GV".oOutput,
                               iIn3Sim := "PF_P10_3_ETDF_TURB_GV".oSim,
                               iText3 := 'Def Ventil  P10.3',
                               iIn4 := "COM_IL_DEF_NON_PRIO1_AGBT2".oOutput,
                               iIn4Sim := "COM_IL_DEF_NON_PRIO1_AGBT2".oSim,
                               iText4 := 'Def Ventil  P1-P9',
                               iEnableP2And := FALSE,
                               iIn5 := "PF_P8_DEF_OH_DEGIV".oOutput,
                               iIn5Sim := "PF_P8_DEF_OH_DEGIV".oSim,
                               iText5 := 'Def RES Dégic P8',
                               iIn6 := 0,
                               iIn6Sim := 0,
                               iEnableNegIn6 := 0,
                               iIn7 := 0,
                               iIn7Sim := 0,
                               iEnableNegIn7 := 0,
                               iIn8 := 0,
                               oOutput => "COM_864083-864079".Def_Non_Prio_AGBT2);
   END_IF;
END_REGION

REGION Network 7: Echange avec API SDM
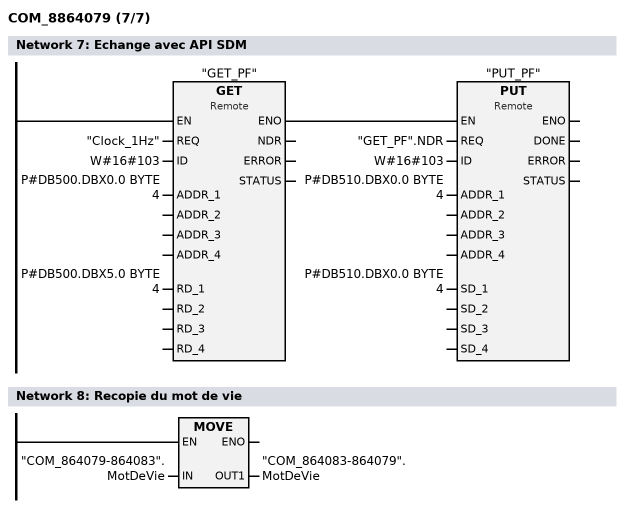
   RUNG wire#powerrail
      { S7_Templates := "[remote_type := Remote, local_type := Variant]" } "GET_PF".GET(REQ := "Clock_1Hz", ID := W#16#103, ADDR_1 := P#DB500.DBX0.0 BYTE 4, ADDR_2 :=, ADDR_3 :=, ADDR_4 :=, RD_1 := P#DB500.DBX5.0 BYTE 4, RD_2 :=, RD_3 :=, RD_4 :=, NDR =>, ERROR =>, STATUS =>)
      { S7_Templates := "[remote_type := Remote, local_type := Variant]" } "PUT_PF".PUT(REQ := "GET_PF".NDR, ID := W#16#103, ADDR_1 := P#DB510.DBX0.0 BYTE 4, ADDR_2 :=, ADDR_3 :=, ADDR_4 :=, SD_1 := P#DB510.DBX0.0 BYTE 4, SD_2 :=, SD_3 :=, SD_4 :=, DONE =>, ERROR =>, STATUS =>)
   END_RUNG
   // the same network as SCL:
   "GET_PF"(REQ := "Clock_1Hz",   // GET
            ID := W#16#103,
            ADDR_1 := P#DB500.DBX0.0 BYTE 4,
            RD_1 := P#DB500.DBX5.0 BYTE 4,
            ENO => #_w1);
   IF #_w1 THEN
       "PUT_PF"(REQ := "GET_PF".NDR, ID := W#16#103, ADDR_1 := P#DB510.DBX0.0 BYTE 4, SD_1 := P#DB510.DBX0.0 BYTE 4);   // PUT
   END_IF;
END_REGION

REGION Network 8: Recopie du mot de vie
   RUNG wire#powerrail
      { S7_GenerateENO := "TRUE" } Move(in := "COM_864079-864083".MotDeVie, out1 => "COM_864083-864079".MotDeVie)
   END_RUNG
   // the same network as SCL:
   "COM_864083-864079".MotDeVie := "COM_864079-864083".MotDeVie;
END_REGION
END_FUNCTION
